FUNCTION F_Loops : INT 
VAR_INPUT
	nInputNum1 : INT;
END_VAR
VAR_OUTPUT
	nResult1 : INT;
	nResult2 : INT;
	nResult3 : INT;
END_VAR
VAR
	nCounter : INT;
END_VAR

FOR nCounter := 1 TO nInputNum1 DO
	nResult1 := nResult1 + nCounter;
END_FOR

nInputNum1 := 1;
WHILE nInputNum1 <> 10 DO
	nInputNum1 := nInputNum1 + 1;
	nResult2 := nResult2 + nInputNum1;
END_WHILE

nCounter := 0;
REPEAT
	nCounter := nCounter + 1;
	nResult3 := nResult3 + nCounter;
	
	UNTIL
	nCounter = 10
END_REPEAT

END_FUNCTION

(* stored: Version 1.1.0.1, ProductVersion 3.1.4024.16
   POU F_Loops: Id {4d37c3f4-a82b-4abe-9268-884651b5e606}, SpecialFunc None *)
